(* IEC 61131-3 sources: 2026_Projet_YGO_ExcavatriceDragage/CODE/CODEURS, 10 files *)

(* ---- ST_Encoder_Calib.st ---- *)
(* ═══════════════════════════════════════════════════════════════
   🧲 ST_Encoder_Calib — Calibration & référence codeur (1 par treuil, RETAIN)
   ───────────────────────────────────────────────────────────────
   📄 Doc métier : DOC/AF/AF_Partie-09_Fonction_Encoder_v2.1.md
                   DOC/AF/AF_Partie-03_Contrats_Composants_v2.1.md
   🎛️ Une instance RETAIN par treuil (M1_EncoderCalib / M2_EncoderCalib).
   ═══════════════════════════════════════════════════════════════ *)

TYPE ST_Encoder_Calib :
STRUCT
    HomingRefRaw                  : UDINT;   // Valeur brute figée au dernier homing réussi
    LastKnownRawPos                : UDINT;   // Dernier point brut valide connu (§3.7, continu)
    RestartCoherenceTolerancePts    : UDINT := 1000;  // Tolérance redémarrage (~12% PointsPerRev 8192)
    Homed                          : BOOL;    // TRUE dès qu'un référencement a réussi
    HomingSuspect                  : BOOL;    // TRUE si incohérence détectée au redémarrage (§3.7)
END_STRUCT
END_TYPE

(* ---- ST_EncoderCalib.st ---- *)
(* ═══════════════════════════════════════════════════════════════
   🧲 ST_EncoderCalib — Calibration/référence codeur (1 par treuil, RETAIN)
   ───────────────────────────────────────────────────────────────
   📄 Doc métier : DOC/AF_Partie-09_Fonction_Encoder_Homing_v2.0.md §9
   🎛️ Une instance RETAIN par treuil (M1_EncoderCalib / M2_EncoderCalib).
   ⚠️ Ce lot (acquisition + mise à l'échelle) : `HomingRefRaw` reste
      modifiable MANUELLEMENT (RETAIN, valeur de test) tant que
      `FB_Encoder_Homing` (qui l'écrit normalement, §5) n'est pas codé —
      même principe que le stub GVL du lot Winch.
   ═══════════════════════════════════════════════════════════════ *)

TYPE ST_EncoderCalib :
STRUCT
    HomingRefRaw                  : UDINT;   // Valeur brute figée au dernier homing réussi
    LastKnownRawPos                : UDINT;   // Dernier point brut valide connu (§3.7, continu)
    RestartCoherenceTolerancePts    : UDINT := 1000;  // Tolérance redémarrage (~12% PointsPerRev 8192)
    Homed                          : BOOL;    // TRUE dès qu'un référencement a réussi
    HomingSuspect                  : BOOL;    // TRUE si incohérence détectée au redémarrage (§3.7)
END_STRUCT
END_TYPE

(* ---- ST_EncoderMeasurement.st ---- *)
(* ═══════════════════════════════════════════════════════════════
   📏 ST_EncoderMeasurement — Mesures codeur qualifiées (1 sous-DUT par treuil)
   ───────────────────────────────────────────────────────────────
   📄 Lot M1 · Doc : DOC/AF_Partie-06_Acquisition_Qualification_IO_v2.0.md §2ter
   🎨 Facts de la chaîne de mesure pure : Abs → Scale → Safety → SpeedMeasure.
   🔗 Producteur : PRG_02_Acquisition_CFC (chaîne codeur du treuil concerné).
   ✅ Tout BOOL = TRUE état normalisé. Aucun brut EtherCAT (alarmes/warnings,
      DEVICE_STATE) : ils restent exposés via ST_EncoderHMI (Supervision).
   ═══════════════════════════════════════════════════════════════ *)
TYPE ST_EncoderMeasurement :
STRUCT
    RawPos           : UDINT; (* Position brute codeur — gelée si EncoderAvailable=FALSE *)
    EncoderAvailable : BOOL;  (* TRUE = bus/esclave opérationnel *)
    CablePosM        : REAL;  (* Position câble (m, signée, + enroulé) *)
    CablePosMSafe    : REAL;  (* Position câble bornée [-99;+99] m — gelée sur doute *)
    EncoderIncoherent: BOOL;  (* TRUE = incohérence redémarrage → refuse SEMI_AUTO *)
    Speed_Mps        : REAL;  (* Vitesse absolue (m/s) — 0.0 si SpeedValid=FALSE *)
    SignedSpeed_Mps  : REAL;  (* Vitesse signée (m/s, + montée) — 0.0 si SpeedValid=FALSE *)
    SpeedValid       : BOOL;  (* TRUE si ≥ 6 éch. couvrant 50 ms *)
END_STRUCT
END_TYPE

(* ---- ST_EncoderMeasurements.st ---- *)
(* ═══════════════════════════════════════════════════════════════
   📏 ST_EncoderMeasurements — Mesures codeurs M1/M2 (contrat frontière)
   ───────────────────────────────────────────────────────────────
   📄 Lot M1 · Doc : DOC/AF/AF_Partie-06_Acquisition_Qualification_IO_v2.1.md §2ter
   🎨 Un sous-DUT par treuil (M1, M2) de la chaîne de mesure pure.
   🔗 Producteur unique : PRG_02_Acquisition_CFC (rang 02, chaîne codeur M1/M2).
      Lecteurs : PRG_04_Treuils_Benne_CFC, PRG_03_Modes_Cycle_CFC, Supervision/IHM.
   🛡️ Sans simulation : M1 reflète COD1, M2 reflète COD2 — jamais croisés.
   ═══════════════════════════════════════════════════════════════ *)
TYPE ST_EncoderMeasurements :
STRUCT
    M1 : ST_EncoderMeasurement; (* Chaîne de mesure treuil M1 (COD1) *)
    M2 : ST_EncoderMeasurement; (* Chaîne de mesure treuil M2 (COD2) *)
END_STRUCT
END_TYPE

(* ---- FB_Encoder_Abs.st ---- *)
(* ═══════════════════════════════════════════════════════════════
   🧲 FB_Encoder_Abs — Acquisition codeur absolu (accès bus, 1 responsabilité)
   ───────────────────────────────────────────────────────────────
   📄 Doc métier : DOC/AF_Partie-09_Fonction_Encoder_Homing_v2.0.md §3/§6
   ⚠️ RÉÉCRITURE COMPLÈTE (remplace la version legacy du projet, dossier
      CODEUR) : l'ancienne version utilisait `HomingTrigger` (recalage
      instantané par simple offset) + un mode `Teach` auto-calibré —
      **incompatibles** avec le design Partie10 (preset SDO avec
      accusé, formule `CableM_PerRev` fixe). Retirés : `HomingTrigger`,
      `WaterLevelOffset`, `TeachActive/StartRaw/EndRaw/RealDistance`.
   🧩 1 FB = 1 responsabilité : accès bus EtherCAT + séquence d'écriture
      preset. N'orchestre PAS le homing lui-même (ça sera le rôle de
      `FB_Encoder_Homing`, pas codé ce lot) — `PresetRequest`/`PresetValue`
      sont pilotés en dur (`FALSE`/`0`) dans `PRG_MAIN` pour l'instant.
   🧊 Principe « geler sur doute » (§6) : `RawPos`/`AngleRaw`/`TurnCount`
      ne sont PAS mis à jour si `EncoderAvailable = FALSE` — ils
      conservent leur dernière valeur plausible.
   ✅ SÉQUENCE PRESET (§5) — CONFIRMÉ TERRAIN 2026-07-02 : `PresetTriggerCmd := 2`
      (valeur de commande, pas un masque de bits) déclenche le
      référencement du codeur à `PresetValueOut`. `CodeSeqTriggerCmd`
      (canal réel `COD1_CodeSeqTrigCmd`) reste `0`, rôle **non identifié**
      (même par l'utilisateur/terrain) — ne jamais lui donner une valeur
      arbitraire tant que sa fonction n'est pas confirmée.
   🔴 PERTE DE FONCTION SIGNALÉE : l'ancienne version composait
      `FB_Encoder_Safety` en interne (survitesse via `In_SpdValue`).
      Ce n'est PAS repris ici (Partie10 ne le demande pas, hors
      périmètre du document) — `FB_Encoder_Safety` (overspeed) devient
      orphelin tant qu'un lot dédié ne décide pas de son sort (fusion
      avec le "saut incohérent" Partie10 §3.5, ou reprise telle quelle).
   🔧 CORRECTIF (2026-07-03, retour terrain) : `InvertDirection` **retiré**.
      Confirmé terrain : l'objet CoE `6000h` (bit0 : 4→5) inverse le sens
      de comptage **côté codeur** (F58x8 Kübler), configuré en **Startup
      Parameter** CODESYS (init automate) — pas un paramètre PLC. L'ancien
      calcul logiciel (`16#FFFFFFFF - RawPosIn`) était de toute façon
      **buggé** : il inversait sur toute la plage `UDINT` (32 bits) au
      lieu de la plage réelle du codeur (25 bits, `PointsPerRev ×
      MultiTurnRevsMax`), produisant des positions incohérentes après
      homing. Voir Partie10 §3bis.
   ═══════════════════════════════════════════════════════════════ *)

// === DECLARATION (à coller dans la partie déclaration du POU FB_Encoder_Abs) ===

FUNCTION_BLOCK PUBLIC FB_Encoder_Abs
VAR_INPUT
    Enable              : BOOL;        // Standard
    Reset               : BOOL;        // Acquittement défaut (front)
    PowerContactorEngaged     : BOOL;        // Standard
    Mode                : E_Mode;      // Standard (contexte, pas encore exploité ce lot)
    RawPosIn            : UDINT;       // Brut EtherCAT (ex. COD1_PosValue, %ID)
    AlarmsIn            : UINT;        // Brut EtherCAT (ex. COD1_Alarms)
    WarningsIn          : UINT;        // Brut EtherCAT (ex. COD1_Warnings) — informatif seulement
    SlaveOperational    : BOOL;        // FB_DiagEthercat — esclave EtherCAT opérationnel
    PointsPerRev        : UDINT := 8192;  // Résolution codeur confirmée (Partie10 §3.3)
    PresetRequest       : BOOL;        // Front — piloté par FB_Encoder_Homing via PRG_02_Encoders
    PresetValue         : UDINT;       // Cible brute — piloté par FB_Encoder_Homing (stub 0 ce lot)
    PresetTimeout       : TIME := T#2s;
    PresetTolerancePts  : UDINT := 10; // Tolérance relecture post-preset
END_VAR
VAR_OUTPUT
    Ready               : BOOL;
    Busy                : BOOL;
    Done                : BOOL;
    Error               : BOOL;
    ErrorId             : WORD;        // bit0: "Défaut communication codeur" - alarme/bus codeur ; bit1: "Erreur référencement (timeout)" - preset refusé/timeout
    State               : E_State;
    StateAtError        : E_State;
    RawPos              : UDINT;       // Position brute — GELÉE si EncoderAvailable=FALSE
    EncoderAvailable    : BOOL;
    AngleRaw            : UINT;        // Informatif maintenance : RawPos MOD PointsPerRev
    TurnCount           : UDINT;       // Informatif maintenance : RawPos / PointsPerRev
    PresetAck           : BOOL;        // Pulse 1 cycle — écriture confirmée
    PresetNak           : BOOL;        // Pulse 1 cycle — écriture refusée/timeout
    PresetTriggerCmd    : WORD;        // → à câbler sur COD_PresettTrigCmd (RxPDO)
    CodeSeqTriggerCmd   : WORD;        // → à câbler sur COD_CodeSeqTrigCmd (RxPDO)
    PresetValueOut      : UDINT;       // → à câbler sur COD_PresetValue (RxPDO)
END_VAR
VAR
    ResetEdge           : R_TRIG;
    ErrorEdge           : R_TRIG;
    PresetReqEdge       : R_TRIG;
    PresetTimer         : TON;
    PresetSeqStep       : INT;         // 0=IDLE, 1=pulse CodeSeq, 2=pulse Trig, 3=attente confirmation
    RawDiff             : DINT;
    PresetTimerVisual   : TON;         // Timer pour laisser le temps de voir l'impulsion (1.5s)
END_VAR

// === IMPLEMENTATION (à coller dans le corps ST du POU FB_Encoder_Abs) ===

// 🛑 1. GATE
IF NOT Enable THEN
    EncoderAvailable := FALSE;
    State := E_State.DISABLED;
    Ready := FALSE; Busy := FALSE; Done := FALSE;
    PresetTriggerCmd := 16#0000; CodeSeqTriggerCmd := 16#0000; PresetValueOut := 0;
    PresetSeqStep := 0;
    PresetTimer(IN := FALSE, PT := PresetTimeout);
    PresetTimerVisual(IN := FALSE, PT := T#500MS);
    RETURN;
END_IF;

Ready := TRUE;
State := E_State.READY;

// 🔑 2. RESET FRONT
ResetEdge(CLK := Reset);

// 🔍 3. DIAGNOSTIC BUS / ALARME
IF (AlarmsIn <> 0) OR NOT SlaveOperational THEN
    ErrorId := ErrorId OR 16#0001;
ELSE
    ErrorId := ErrorId AND 16#FFFE; (* Auto-clearing dès que le bus et l'esclave sont OK *)
END_IF;
EncoderAvailable := (ErrorId AND 16#0001) = 0;

// 📥 4. LECTURE POSITION — GELER SUR DOUTE (Partie10 §6)
// Si EncoderAvailable=FALSE : RawPos/AngleRaw/TurnCount conservent leur dernière valeur (pas de RETURN
// global ici pour ne pas geler aussi la séquence preset/l'état — seule la lecture est gelée).
IF EncoderAvailable THEN
    RawPos := RawPosIn;   // 🔧 2026-07-03 : sens de comptage géré côté codeur (CoE 6000h bit0,
                          // startup parameter CODESYS) — voir Partie10 §3bis. Plus de calcul ici.
    AngleRaw := UDINT_TO_UINT(RawPos MOD PointsPerRev);
    TurnCount := RawPos / PointsPerRev;
END_IF;

// 🔧 5. SÉQUENCE PRESET (écriture bus)
// ✅ Confirmé terrain (2026-07-02) : PresettTrigCmd := 2 déclenche le référencement à
//    PresetValue (valeur de commande, pas un masque de bits — corrige l'hypothèse initiale).
// 🔴 CodeSeqTrigCmd : rôle NON identifié (même par l'utilisateur/terrain) — laissé à 0,
//    PAS piloté tant que sa fonction n'est pas confirmée (fiche technique ou essai dédié).
//    Ne jamais lui donner une valeur arbitraire "au cas où".
PresetReqEdge(CLK := PresetRequest);
PresetAck := FALSE; PresetNak := FALSE; // pulses 1 cycle uniquement
CodeSeqTriggerCmd := 16#0000;           // 🔴 non piloté — rôle inconnu, voir note ci-dessus
CASE PresetSeqStep OF
    0: // IDLE
        PresetTriggerCmd := 0;
        IF PresetReqEdge.Q AND EncoderAvailable THEN
            PresetValueOut := PresetValue;
            PresetSeqStep := 1;
            PresetTimer(IN := TRUE, PT := PresetTimeout);
        END_IF;
    1: // Déclenchement preset (laissé actif pendant 0.5s pour confort visuel en simulation/bus)
        PresetTriggerCmd := 2;   // ✅ Valeur confirmée terrain — référence le codeur à PresetValueOut
        RawDiff := UDINT_TO_DINT(RawPos) - UDINT_TO_DINT(PresetValueOut);
        IF ABS(RawDiff) <= UDINT_TO_DINT(PresetTolerancePts) THEN
            PresetTimer(IN := FALSE, PT := PresetTimeout);
            PresetTimerVisual(IN := TRUE, PT := T#500MS);
            IF PresetTimerVisual.Q THEN
                PresetTriggerCmd := 0;
                PresetAck := TRUE;
                PresetSeqStep := 0;
                PresetTimerVisual(IN := FALSE, PT := T#500MS);
            END_IF;
        ELSIF PresetTimer.Q THEN
            PresetTriggerCmd := 0;
            PresetNak := TRUE;
            ErrorId := ErrorId OR 16#0002;
            PresetSeqStep := 0;
            PresetTimer(IN := FALSE, PT := PresetTimeout);
            PresetTimerVisual(IN := FALSE, PT := T#500MS);
        END_IF;
END_CASE;
IF ResetEdge.Q AND (PresetSeqStep = 0) THEN
    ErrorId := ErrorId AND 16#FFFD;
END_IF;

// 🧾 6. ERROR / STATEATERROR
Error := (ErrorId <> 16#0000);
ErrorEdge(CLK := Error);
IF ErrorEdge.Q THEN
    StateAtError := State;
END_IF;

Busy := (PresetSeqStep <> 0);
Done := PresetAck;

(* ---- FB_Encoder_Homing.st ---- *)
(* ═══════════════════════════════════════════════════════════════
   🎯 FB_Encoder_Homing — Référencement codeur nominal ou unitaire MAINT_N2
   ───────────────────────────────────────────────────────────────
   📄 Doc métier : DOC/AF_Partie-09_Fonction_Encoder_Homing_v2.0.md §1/§5/§7bis
   ⚠️ PÉRIMÈTRE : flux nominal (capteur haut + cible paramétrable) ou
      unitaire MAINT_N2 (treuil sélectionné + cible libre). Aucun mouvement
      moteur n'est piloté ici.
   🔌 PAS un FB de mouvement (Partie3 §1bis) : il n'écrit qu'une valeur
      de calibration, le treuil étant déjà à l'arrêt confirmé. Pas de
      `StartStop`/`SafeStop`.
   🧮 Calcul (généralise le cas historique cible=0.00, Partie10 §3.2/§3.3) :
      - `PresetValue` = `HomingRefTargetNominal` = (PointsPerRev × MultiTurnRevsMax) / 2
        (constante, TOUJOURS la même — centre exact de la plage, marge anti-débordement)
      - `HomingRefRaw` = `PresetValue` − round(`CfgTopSensorPosM` × PointsPerRev / CableM_PerRev)
        (ainsi `CablePosM` = `CfgTopSensorPosM` exactement au moment du homing)
      ⚠️ ÉVOLUTION vs interface §5 d'origine : `HomingRefRaw` est ajouté en sortie explicite
      (le document original supposait implicitement `HomingRefRaw := PresetValue`, valable
      uniquement pour une cible à 0.00 — ne fonctionne plus avec une cible non nulle ≈8.50 m).
   🧊 `ST_EncoderCalib` géré en interne (`VAR RETAIN`) — expose `Homed`/`HomingSuspect`/
      `HomingRefRaw` en sortie pour les consommateurs (`FB_Encoder_Scale`).
   🔴 SIMPLIFICATIONS assumées pour ce lot (à documenter/lever plus tard si besoin) :
      - Les 2 instances (M1/M2) sont autonomes : le même bouton IHM pilote les deux `Home`
        simultanément (câblage PRG_MAIN), mais chacune valide/rejette SES PROPRES conditions
        indépendamment (pas d'attente mutuelle ni de synchro de déclenchement).
      - `BtnConfirmCoherence`/§3.7 (incohérence redémarrage) : implémenté a minima (bit9), mais
        non testé en conditions réelles de coupure secteur — à revalider.
   ═══════════════════════════════════════════════════════════════ *)

// === DECLARATION (à coller dans la partie déclaration du POU FB_Encoder_Homing) ===

FUNCTION_BLOCK PUBLIC FB_Encoder_Homing
VAR_INPUT
    Enable               : BOOL;        // Standard
    Reset                : BOOL;        // Acquittement défaut (front) — bits 0/2/3/4/5 (voir §ErrorId)
    PowerContactorEngaged      : BOOL;        // Standard
    Mode                 : E_Mode;      // MAINT_N1 requis pour le flux nominal
    Home                 : BOOL;        // Demande de référencement (front, bouton IHM UNIQUE)
    UnitaryMode          : BOOL;        // TRUE = flux unitaire à cible libre (MAINT_N2 uniquement)
    WinchSelected        : BOOL;        // TRUE = cette instance est le treuil sélectionné
    CfgHomingTargetM        : REAL;        // Cible libre unitaire, limitée à [-99.0 ; +99.0] m
    BtnConfirmCoherence     : BOOL;        // Front — lève le doute §3.7 (bit9), sans réhoming complet
    TopPositionSensor    : BOOL;        // 🔧 2026-07-02 : capteur position haute UNIQUE, COMMUN aux 2 treuils
                                         // (les 2 câbles hissent ensemble le même ensemble mécanique) — câblé
                                         // IDENTIQUEMENT sur les instances M1 ET M2 (PAS un capteur par treuil),
                                         // voir PRG_MAIN.st
    CfgTopSensorPosM   : REAL := 8.5;   // Cible homing nominal (RETAIN site, voir Partie10 §7bis)
    FwdRevSpeedFeedbackOff : BOOL;      // 🔧 REX 2026-07-07 : retour unique "tous contacteurs sens+vitesse
                                         // retombés" CE TREUIL — arrêt confirmé (remplace ContactorFeedbackFwd/Rev)
    BrakeFeedback        : BOOL;        // Retour contacteur frein CE TREUIL (TRUE = relâché, FALSE = collé)
    RawPos               : UDINT;       // Sortie FB_Encoder_Abs (déjà gelée sur doute)
    EncoderAvailable     : BOOL;        // Sortie FB_Encoder_Abs
    PresetAck            : BOOL;        // Pulse — sortie FB_Encoder_Abs (écriture confirmée)
    PresetNak            : BOOL;        // Pulse — sortie FB_Encoder_Abs (écriture refusée/timeout)
    PointsPerRev         : UDINT := 8192;   // Confirmé fiche technique (Partie10 §3.3)
    MultiTurnRevsMax     : UDINT := 4096;   // Confirmé fiche technique (Partie10 §3.3)
    CableM_PerRev        : REAL := 2.0;     // Confirmé terrain 2026-07-02 (Partie10 §2)
    BypassGlobal         : BOOL := FALSE;   // 🌐 Ignore arrêt confirmé et capteur haut (mise en service)
END_VAR
VAR_OUTPUT
    Ready                : BOOL;
    Busy                 : BOOL;
    Done                 : BOOL;        // Pulse 1 cycle — référencement réussi (miroir PresetAck)
    Error                : BOOL;
    ErrorId              : WORD;        // Voir table de bits en en-tête de fichier / doc §5
    State                : E_State;
    StateAtError         : E_State;
    PresetRequest        : BOOL;        // Pulse → FB_Encoder_Abs.PresetRequest
    PresetValue          : UDINT;       // → FB_Encoder_Abs.PresetValue (= HomingRefTargetNominal)
    Homed                : BOOL;        // RETAIN interne, miroir Calib.Homed
    HomingSuspect        : BOOL;        // RETAIN interne, miroir Calib.HomingSuspect
    HomingRefRaw         : UDINT;       // RETAIN interne, miroir Calib.HomingRefRaw → FB_Encoder_Scale
END_VAR
VAR_IN_OUT
    Calib                : ST_EncoderCalib;   // Référence vers l'état persistant global (survit aux téléchargements)
END_VAR
VAR
    ResetEdge            : R_TRIG;
    ErrorEdge            : R_TRIG;
    HomeEdge             : R_TRIG;
    ConfirmCoherenceEdge : R_TRIG;
    InitDone             : BOOL;        // Contrôle cohérence §3.7 fait une fois par session Enable
    ArretConfirme        : BOOL;
    PresetValueCalc      : UDINT;       // = HomingRefTargetNominal (constant tant que PointsPerRev/MultiTurnRevsMax fixes)
    TargetPoints         : DINT;        // Écart signé CfgTopSensorPosM → points, figé pendant la séquence
    TargetPositionM      : REAL;        // Cible retenue : nominale ou unitaire
    RawDiffRestart       : DINT;        // Écart |RawPos - LastKnownRawPos| au redémarrage (§3.7)
END_VAR

// === IMPLEMENTATION (à coller dans le corps ST du POU FB_Encoder_Homing) ===

// 🛑 1. GATE — neutralisation ; on continue toutefois d'exposer le dernier état RETAIN connu
// (FB_Encoder_Scale a besoin de HomingRefRaw même si ce FB est désactivé)
IF NOT Enable OR NOT PowerContactorEngaged THEN
    PresetRequest := FALSE;
    PresetValue := 0;
    State := E_State.DISABLED;
    Ready := FALSE; Busy := FALSE; Done := FALSE;
    InitDone := FALSE;   // Force un nouveau contrôle §3.7 à la prochaine activation
    Homed := Calib.Homed;
    HomingSuspect := Calib.HomingSuspect;
    HomingRefRaw := Calib.HomingRefRaw;
    RETURN;
END_IF;

Ready := TRUE;

// 🔑 2. FRONTS
ResetEdge(CLK := Reset);
HomeEdge(CLK := Home);
ConfirmCoherenceEdge(CLK := BtnConfirmCoherence);

// 🔍 3. COHÉRENCE AU REDÉMARRAGE (§3.7) — une fois par session Enable, dès que le codeur répond
IF NOT InitDone THEN
    State := E_State.INIT;
    IF EncoderAvailable THEN
        RawDiffRestart := UDINT_TO_DINT(RawPos) - UDINT_TO_DINT(Calib.LastKnownRawPos);
        IF Calib.Homed AND (ABS(RawDiffRestart) > UDINT_TO_DINT(Calib.RestartCoherenceTolerancePts)) THEN
            Calib.HomingSuspect := TRUE;
            ErrorId := ErrorId OR 16#0200;   // bit9 : incohérence codeur au redémarrage
        END_IF;
        InitDone := TRUE;
    END_IF;
ELSE
    IF State = E_State.INIT THEN State := E_State.READY; END_IF;
END_IF;

// ✅ 4. LEVÉE DU DOUTE (BtnConfirmCoherence, §3.7) — indépendant du Reset générique
IF ConfirmCoherenceEdge.Q AND (Mode = E_Mode.MAINT_N1 OR Mode = E_Mode.MAINT_N2) THEN
    Calib.HomingSuspect := FALSE;
    ErrorId := ErrorId AND 16#FDFF;   // efface bit9
END_IF;

// 🎯 5. DEMANDE DE RÉFÉRENCEMENT (flux nominal)
// 🛡️ Les cibles nominale et unitaire sont rejetées hors du domaine codeur sûr [-99.00;+99.00] m.
// 🔧 REX 2026-07-07 : FwdRevSpeedFeedbackOff remplace (NOT ContactorFeedbackFwd) AND (NOT ContactorFeedbackRev)
// 🌐 BypassGlobal = TRUE → on saute la vérification d'arrêt (mise en service)
ArretConfirme := BypassGlobal OR (FwdRevSpeedFeedbackOff AND BrakeFeedback);

PresetRequest := FALSE;   // Défaut chaque cycle — repose uniquement sur le front HomeEdge ci-dessous
IF HomeEdge.Q AND (State <> E_State.BUSY) THEN
    IF UnitaryMode THEN
        TargetPositionM := CfgHomingTargetM;
    ELSE
        TargetPositionM := CfgTopSensorPosM;
    END_IF;

    // ✅ Homing autorisé en MAINT_N1 et MAINT_N2 — interdit en SEMI_AUTO et en cycle AUTO
    // 🌐 BypassGlobal = TRUE → saute TOUTES les vérifications, force le homing
    IF BypassGlobal THEN
        // Force homing sans condition
        PresetValueCalc := (PointsPerRev * MultiTurnRevsMax) / 2;
        TargetPoints := REAL_TO_DINT(TargetPositionM * UDINT_TO_REAL(PointsPerRev) / CableM_PerRev);
        PresetValue := PresetValueCalc;
        PresetRequest := TRUE;
        State := E_State.BUSY;
    ELSIF (Mode <> E_Mode.MAINT_N1) AND (Mode <> E_Mode.MAINT_N2) THEN
        ErrorId := ErrorId OR 16#0001;        // bit0 : mode non autorisé (seulement MAINT N1/N2)
    ELSIF UnitaryMode AND (Mode <> E_Mode.MAINT_N2) THEN
        ErrorId := ErrorId OR 16#0001;
    ELSIF UnitaryMode AND NOT WinchSelected THEN
        ErrorId := ErrorId OR 16#0002;        // bit1 : mauvais treuil sélectionné
    ELSIF NOT EncoderAvailable THEN
        ErrorId := ErrorId OR 16#0008;        // bit3 : codeur indisponible
    ELSIF NOT ArretConfirme THEN
        ErrorId := ErrorId OR 16#0004;        // bit2 : arrêt non confirmé (contacteurs/frein)
    ELSIF (TargetPositionM < -99.0) OR (TargetPositionM > 99.0) THEN
        ErrorId := ErrorId OR 16#0010;        // bit4 : cible nominale/unitaire hors limites
    ELSIF NOT BypassGlobal AND NOT UnitaryMode AND (TargetPositionM <> 0.0) AND TopPositionSensor THEN
        ErrorId := ErrorId OR 16#0010;        // bit4 : capteur position haute non confirmé
    ELSE
        // ✅ Toutes conditions réunies : calcul de la cible brute et déclenchement
        ErrorId := ErrorId AND 16#FFC0;       // Nettoie les erreurs de rejet 0..5
        PresetValueCalc := (PointsPerRev * MultiTurnRevsMax) / 2;               // Centre exact (§3.3)
        TargetPoints := REAL_TO_DINT(TargetPositionM * UDINT_TO_REAL(PointsPerRev) / CableM_PerRev);
        PresetValue := PresetValueCalc;
        PresetRequest := TRUE;                // Pulse 1 cycle — FB_Encoder_Abs détecte le front lui-même
        State := E_State.BUSY;
    END_IF;
END_IF;

// ⏳ 6. SUIVI DE LA SÉQUENCE (BUSY → confirmation)
Done := FALSE;
IF State = E_State.BUSY THEN
    IF PresetAck THEN
        Calib.HomingRefRaw := DINT_TO_UDINT(UDINT_TO_DINT(PresetValueCalc) - TargetPoints);
        Calib.Homed := TRUE;
        Calib.HomingSuspect := FALSE;
        Calib.LastKnownRawPos := PresetValueCalc;
        Done := TRUE;
        State := E_State.READY;
        // 🔧 REX 2026-07-24 : Un homing réussi efface l'intégralité de ErrorId (y compris les anciens rejets 0..5 et le bit9)
        ErrorId := 16#0000;
    ELSIF PresetNak THEN
        ErrorId := ErrorId OR 16#0020;        // bit5 : preset refusé/timeout (voir FB_Encoder_Abs)
        State := E_State.READY;
    END_IF;
END_IF;

// 🧾 7. RESET (front) — efface les bits « dernière tentative rejetée » (pas de cause persistante
// à revérifier ici : le prochain Home réévalue toutes les conditions de zéro, voir §5)
IF ResetEdge.Q THEN
    ErrorId := ErrorId AND 16#FFC0;   // efface bits 0..5 (garde bit9, levé seulement par BtnConfirmCoherence/Home)
END_IF;

// 📤 8. SORTIES ÉTAT
Error := (ErrorId <> 16#0000);
ErrorEdge(CLK := Error);
IF ErrorEdge.Q THEN
    StateAtError := State;
END_IF;

// Mise à jour continue du point brut valide connu (hors séquence de homing elle-même)
IF EncoderAvailable AND (State <> E_State.BUSY) THEN
    Calib.LastKnownRawPos := RawPos;
END_IF;

Busy := (State = E_State.BUSY);
Homed := Calib.Homed AND NOT Calib.HomingSuspect; // 🆕 REX 2026-07-08 : Perd l'état homed si suspect (démarrage ou fonctionnement), restauré après BtnConfirmCoherence
HomingSuspect := Calib.HomingSuspect;
HomingRefRaw := Calib.HomingRefRaw;

(* ---- FB_Encoder_Safety.st ---- *)
(* ═══════════════════════════════════════════════════════════════
   🛡️ FB_Encoder_Safety — Bornage physique + relais incohérence redémarrage (1 par treuil)
   ───────────────────────────────────────────────────────────────
   📄 Doc métier : DOC/AF_Partie-10_Fonction_Encoder_Homing_v1.10.md §3.6/§3.7
   🔌 FB STANDARD (Partie3 §1bis) : pas un FB de mouvement, pas de StartStop/SafeStop.
   🎯 PÉRIMÈTRE CE LOT (répond à l'incident CablePosM≈4096m après reset RETAIN) :
      - §3.6 Bornage absolu [-99.00 ; +99.00] m : `CablePosM` hors plage → valeur
        jugée IMPOSSIBLE, sortie `CablePosMSafe` GELÉE sur dernière valeur plausible
        (principe « geler sur doute », §6), ErrorId bit0.
      - §3.7 Relais de `HomingSuspect` (déjà détecté par `FB_Encoder_Homing`, jamais
        consommé nulle part avant ce lot) : ErrorId bit1.
      - `EncoderIncoherent` (= Error) → consommé par `FB_Modes` pour REFUSER
        `SEMI_AUTO` (reste possible de travailler en MAINT_N1/N2 pour re-référencer,
        voir échange utilisateur — PAS de SafeStop ici, ne bloque jamais le mouvement).
   🔴 HORS PÉRIMÈTRE CE LOT (Partie10 §3.5, reporté) : détection de saut EN COURS
      D'EXPLOITATION (plausibilité vitesse codeur, calcul sur cycles EtherCAT 4ms) —
      lot dédié à part entière, pas fait ici.
   ═══════════════════════════════════════════════════════════════ *)

// === DECLARATION (à coller dans la partie déclaration du POU FB_Encoder_Safety) ===

FUNCTION_BLOCK PUBLIC FB_Encoder_Safety
VAR_INPUT
    Enable           : BOOL;        // Standard
    Reset            : BOOL;        // Acquittement défaut (front) — bit0 uniquement (bit1 suit HomingSuspect, voir §7bis)
    EmergencyStopOk  : BOOL;        // Standard
    Mode             : E_Mode;      // Standard (contexte, pas encore exploité ce lot)
    CablePosM        : REAL;        // Sortie FB_Encoder_Scale DE CE TREUIL
    HomingSuspect    : BOOL;        // Sortie FB_Encoder_Homing DE CE TREUIL (§3.7, déjà calculé)
    PositionMinM     : REAL := -99.0;  // Bornage physique dur (Partie10 §3.6)
    PositionMaxM     : REAL := 99.0;
END_VAR
VAR_OUTPUT
    Ready            : BOOL;
    Busy             : BOOL;
    Done             : BOOL;
    Error            : BOOL;
    ErrorId          : WORD;        // bit0: "Position câble hors plage" - position hors plage physique ; bit1: "Incohérence position boot" - incohérence redémarrage (miroir HomingSuspect)
    State            : E_State;
    StateAtError     : E_State;
    CablePosMSafe    : REAL;        // CablePosM gelée sur dernière valeur plausible si hors plage
    EncoderIncoherent: BOOL;        // = Error — consommé par FB_Modes (refuse SEMI_AUTO)
END_VAR
VAR
    ResetEdge             : R_TRIG;
    ErrorEdge             : R_TRIG;
    LastPlausibleCablePosM: REAL;
END_VAR

// === IMPLEMENTATION (à coller dans le corps ST du POU FB_Encoder_Safety) ===

// 🛑 1. GATE — expose la dernière valeur plausible connue même désactivé
IF NOT Enable THEN
    Ready := FALSE; Busy := FALSE; Done := FALSE;
    State := E_State.DISABLED;
    CablePosMSafe := LastPlausibleCablePosM;
    EncoderIncoherent := FALSE;
    RETURN;
END_IF;

Ready := TRUE;
State := E_State.READY;

// 🔑 2. RESET FRONT
ResetEdge(CLK := Reset);

// 🔍 3. BORNAGE PHYSIQUE ABSOLU (§3.6) — bit0
IF (CablePosM < PositionMinM) OR (CablePosM > PositionMaxM) THEN
    ErrorId := ErrorId OR 16#0001;
ELSIF ResetEdge.Q THEN
    ErrorId := ErrorId AND 16#FFFE;
END_IF;

// 🔍 4. RELAIS INCOHÉRENCE REDÉMARRAGE (§3.7, calculée par FB_Encoder_Homing) — bit1
// Pas d'acquittement ici : la levée se fait via BtnConfirmCoherence/nouveau Home côté
// FB_Encoder_Homing (source), ce FB ne fait QUE relayer l'information pour FB_Modes.
IF HomingSuspect THEN
    ErrorId := ErrorId OR 16#0002;
ELSE
    ErrorId := ErrorId AND 16#FFFD;
END_IF;

// 🧊 5. GELER SUR DOUTE (§6) — CablePosMSafe ne suit PAS CablePosM si hors plage
IF (ErrorId AND 16#0001) = 16#0000 THEN
    LastPlausibleCablePosM := CablePosM;
END_IF;
CablePosMSafe := LastPlausibleCablePosM;

// 📤 6. SORTIES ÉTAT
Error := (ErrorId <> 16#0000);
ErrorEdge(CLK := Error);
IF ErrorEdge.Q THEN
    StateAtError := State;
END_IF;

EncoderIncoherent := Error;
Busy := FALSE;
Done := FALSE;

(* ---- FB_Encoder_Scale.st ---- *)
(* ═══════════════════════════════════════════════════════════════
   📏 FB_Encoder_Scale — Mise à l'échelle points → mètres (1 par treuil)
   ───────────────────────────────────────────────────────────────
   📄 Doc métier : DOC/AF_Partie-09_Fonction_Encoder_Homing_v2.0.md §2/§3.1
   ⚠️ RÉÉCRITURE (remplace la version legacy) : formule FIXE
      `CablePosM = (RawPos − HomingRefRaw) × (CableM_PerRev/PointsPerRev)`
      — retire le mode `Teach` auto-calibré (`EnableTeach`/`StartTeachPos`/
      `EndTeachPos`/`RealDistMeters`) : `CableM_PerRev` est un paramètre
      RETAIN fixe (site), pas recalculé dynamiquement (Partie10 §2).
   🧮 Arithmétique signée sûre (§3.1) : conversion en DINT AVANT la
      soustraction (jamais soustraire deux UDINT directement — un
      résultat négatif reboucle silencieusement vers ~2³²).
   🧩 Brique de calcul pure — pas de gel/bornage ici : `RawPos` en
      entrée est déjà gelé par `FB_Encoder_Abs` (§6) ; le bornage
      physique absolu [-99;+99] m est la responsabilité de
      `FB_Encoder_Safety` (§3.6, pas dans ce lot), pas de celle-ci.
   ═══════════════════════════════════════════════════════════════ *)

// === DECLARATION (à coller dans la partie déclaration du POU FB_Encoder_Scale) ===

FUNCTION_BLOCK PUBLIC FB_Encoder_Scale
VAR_INPUT
    RawPos          : UDINT;       // Position brute (sortie FB_Encoder_Abs, déjà gelée sur doute)
    HomingRefRaw    : UDINT;       // Référence brute figée au dernier homing (ST_EncoderCalib)
    CableM_PerRev   : REAL := 2.0; // Câble déroulé par tour (périmètre tambour confirmé 2026-07-02, réglable site)
    PointsPerRev    : UDINT := 8192; // Résolution codeur confirmée (Partie10 §3.3)
END_VAR
VAR_OUTPUT
    CablePosM       : REAL;        // Position câble en mètres, signée (+ enroulé, − sous l'eau)
END_VAR
VAR
    RawDiff         : DINT;        // Écart signé RawPos - HomingRefRaw (§3.1)
END_VAR

// === IMPLEMENTATION (à coller dans le corps ST du POU FB_Encoder_Scale) ===

// 🧮 Écart signé sûr : conversion DINT AVANT soustraction (§3.1) — jamais l'inverse
RawDiff := UDINT_TO_DINT(RawPos) - UDINT_TO_DINT(HomingRefRaw);

// 📏 Formule fixe points → mètres (Partie10 §2)
IF PointsPerRev > 0 THEN
    CablePosM := DINT_TO_REAL(RawDiff) * (CableM_PerRev / UDINT_TO_REAL(PointsPerRev));
ELSE
    CablePosM := 0.0;   // Garde division par zéro (PointsPerRev mal configuré)
END_IF;

(* ---- FB_Encoder_SpeedMeasure.st ---- *)
(* ═══════════════════════════════════════════════════════════════
   📐 FB_Encoder_SpeedMeasure — Mesure de vitesse câble horodatée
   ───────────────────────────────────────────────────────────────
   📄 Doc : DOC/AF_Partie-09_Fonction_Encoder_Homing_v2.0.md §3.8
   🛡️ Sécurité : mesure propriétaire de la chaîne codeur ; aucune réaction machine
   🧩 Dépendances : position sûre fournie par FB_Encoder_Safety
   ═══════════════════════════════════════════════════════════════ *)
FUNCTION_BLOCK PUBLIC FB_Encoder_SpeedMeasure
VAR_INPUT
    Enable        : BOOL; // Autorise l'acquisition
    Reset         : BOOL; // Purge immédiate de l'historique
    Position_M    : REAL; // Position câble sûre en mètres
    PositionValid : BOOL; // TRUE si la chaîne codeur garantit la position
END_VAR
VAR_OUTPUT
    Speed_Mps       : REAL; // Vitesse absolue sur la fenêtre horodatée
    SignedSpeed_Mps : REAL; // Vitesse signée : positive montée, négative descente
    Valid           : BOOL; // TRUE après 6 positions couvrant au moins 50 ms
END_VAR
VAR CONSTANT
    WindowTime   : TIME := T#50MS;
    SamplePeriod : TIME := T#10MS;
    SampleCount  : INT := 6;
END_VAR
VAR
    Positions_M : ARRAY[0..5] OF REAL;
    Timestamps  : ARRAY[0..5] OF TIME;
    CurrentTimestamp : TIME;
    LastTimestamp    : TIME;
    ElapsedSinceSample : TIME;
    WindowElapsed      : TIME;
    CollectedSamples   : INT;
    Index              : INT;
    TimestampInitialized : BOOL;
END_VAR

// ⏱️ Horodatage natif : le calcul utilise le temps réellement écoulé, jamais un cycle supposé.
CurrentTimestamp := TIME();

// 🧹 Toute rupture de confiance purge les six positions : aucune ancienne source ne peut contaminer la mesure.
IF NOT Enable OR Reset OR NOT PositionValid THEN
    Speed_Mps := 0.0;
    SignedSpeed_Mps := 0.0;
    Valid := FALSE;
    CollectedSamples := 0;
    TimestampInitialized := FALSE;
    RETURN;
END_IF;

// 🕒 Première position de la nouvelle fenêtre.
IF NOT TimestampInitialized THEN
    Positions_M[0] := Position_M;
    Timestamps[0] := CurrentTimestamp;
    LastTimestamp := CurrentTimestamp;
    CollectedSamples := 1;
    TimestampInitialized := TRUE;
    Speed_Mps := 0.0;
    SignedSpeed_Mps := 0.0;
    Valid := FALSE;
    RETURN;
END_IF;

// 🛡️ Rebouclage de TIME détecté localement : purge sans réutiliser le delta aberrant (indépendant de T88).
IF CurrentTimestamp < LastTimestamp THEN
    Positions_M[0] := Position_M;
    Timestamps[0] := CurrentTimestamp;
    LastTimestamp := CurrentTimestamp;
    CollectedSamples := 1;
    Speed_Mps := 0.0;
    SignedSpeed_Mps := 0.0;
    Valid := FALSE;
    RETURN;
END_IF;

ElapsedSinceSample := CurrentTimestamp - LastTimestamp;

// 🛡️ Delta nul : aucune division et aucun doublon d'échantillon.
IF ElapsedSinceSample <= T#0MS THEN
    RETURN;
END_IF;

// 📥 Six positions espacées d'au moins 10 ms donnent cinq intervalles sur la fenêtre interne de 50 ms.
IF ElapsedSinceSample >= SamplePeriod THEN
    LastTimestamp := CurrentTimestamp;

    IF CollectedSamples < SampleCount THEN
        Positions_M[CollectedSamples] := Position_M;
        Timestamps[CollectedSamples] := CurrentTimestamp;
        CollectedSamples := CollectedSamples + 1;
    ELSE
        FOR Index := 0 TO 4 DO
            Positions_M[Index] := Positions_M[Index + 1];
            Timestamps[Index] := Timestamps[Index + 1];
        END_FOR;
        Positions_M[5] := Position_M;
        Timestamps[5] := CurrentTimestamp;
    END_IF;

    IF CollectedSamples = SampleCount THEN
        // 🛡️ Ordre temporel et durée minimale contrôlés avant toute conversion/division.
        IF Timestamps[5] >= Timestamps[0] THEN
            WindowElapsed := Timestamps[5] - Timestamps[0];
            IF WindowElapsed >= WindowTime THEN
                SignedSpeed_Mps := (Positions_M[5] - Positions_M[0])
                                   / (UDINT_TO_REAL(TIME_TO_UDINT(WindowElapsed)) / 1000.0);
                Speed_Mps := ABS(SignedSpeed_Mps);
                Valid := TRUE;
            ELSE
                Speed_Mps := 0.0;
                SignedSpeed_Mps := 0.0;
                Valid := FALSE;
            END_IF;
        ELSE
            Speed_Mps := 0.0;
            SignedSpeed_Mps := 0.0;
            Valid := FALSE;
            CollectedSamples := 0;
            TimestampInitialized := FALSE;
        END_IF;
    END_IF;
END_IF;

(* ---- FB_Encoder_SpeedMonitor.st ---- *)
(* ═══════════════════════════════════════════════════════════════════════════════
   🔍 FB_Encoder_SpeedMonitor — Détection de variation brusque de vitesse câble
   ═══════════════════════════════════════════════════════════════════════════════
   📄 Brique standard de diagnostic — aucun pilotage moteur, aucun SafeStop.
   🎯 Compare deux mesures successives de vitesse linéaire câble en m/s.
   🧩 Le seuil et la durée de confirmation sont fournis par l'appelant :
      aucun réglage métier n'est figé dans cette brique.
   🛡️ Une variation confirmée pose ErrorId bit0. Le défaut reste mémorisé
      jusqu'à disparition de la cause et acquittement par front Reset.
   ═══════════════════════════════════════════════════════════════════════════════
   📄 Docs : DOC/AF_Partie-09_Fonction_Encoder_Homing_v2.0.md
*)

FUNCTION_BLOCK PUBLIC FB_Encoder_SpeedMonitor
VAR_INPUT
    Enable                     : BOOL;        // Autorise la surveillance
    Reset                      : BOOL;        // Acquittement par front
    PowerContactorEngaged            : BOOL;        // Contexte sécurité global valide
    Mode                       : E_Mode;      // Contexte de fonctionnement
    SpeedMps                   : REAL;        // Vitesse linéaire absolue mesurée (m/s)
    SpeedVariationThresholdMps : REAL;        // Variation minimale à surveiller (m/s)
    SpeedVariationTimeout      : TIME;        // Durée minimale de confirmation
    SpeedStabilityTimeout      : TIME;        // Durée sans variation avant vitesse stable
END_VAR
VAR_OUTPUT
    Ready                  : BOOL;
    Busy                   : BOOL;
    Done                   : BOOL;
    Error                  : BOOL;
    ErrorId                : WORD;        // bit0 : variation vitesse confirmée
    State                  : E_State;
    StateAtError           : E_State;
    SpeedDeltaMps          : REAL;        // Écart absolu entre deux mesures (m/s)
    SpeedVariationDetected : BOOL;        // Seuil dépassé sur le cycle courant
    SpeedVariationConfirmed: BOOL;        // Seuil dépassé pendant la durée requise
    SpeedStable            : BOOL;        // Vitesse stable pendant SpeedStabilityTimeout
END_VAR
VAR
    ResetEdge          : R_TRIG;
    ErrorEdge          : R_TRIG;
    VariationTimer     : TON;
    StabilityTimer     : TON;
    PreviousSpeedMps   : REAL;
    HasPreviousSpeed   : BOOL;
    VariationActive    : BOOL;
END_VAR

// 🛑 1. GATE — désactivation ou AU non réarmé : aucune alarme persistante.
IF NOT Enable OR NOT PowerContactorEngaged THEN
    Ready := FALSE;
    Busy := FALSE;
    Done := FALSE;
    Error := FALSE;
    ErrorId := 16#0000;
    State := E_State.DISABLED;
    SpeedDeltaMps := 0.0;
    SpeedVariationDetected := FALSE;
    SpeedVariationConfirmed := FALSE;
    SpeedStable := FALSE;
    VariationActive := FALSE;
    HasPreviousSpeed := FALSE;
    VariationTimer(IN := FALSE, PT := SpeedVariationTimeout);
    StabilityTimer(IN := FALSE, PT := SpeedStabilityTimeout);
    RETURN;
END_IF;

Ready := TRUE;
Busy := FALSE;
Done := FALSE;
State := E_State.READY;

// 🔑 2. RESET FRONT — l'acquittement n'efface le défaut que si la cause a disparu.
ResetEdge(CLK := Reset);

// 📏 3. CALCUL DE L'ÉCART DE VITESSE — première mesure utilisée comme référence.
IF NOT HasPreviousSpeed THEN
    PreviousSpeedMps := SpeedMps;
    HasPreviousSpeed := TRUE;
    SpeedDeltaMps := 0.0;
ELSE
    SpeedDeltaMps := ABS(SpeedMps - PreviousSpeedMps);
    PreviousSpeedMps := SpeedMps;
END_IF;

// 🔍 4. DÉTECTION BRUTE + FILTRE TEMPOREL — pas de déclenchement si la durée vaut zéro.
VariationActive := HasPreviousSpeed
                   AND (SpeedVariationThresholdMps >= 0.0)
                   AND (SpeedVariationTimeout > T#0ms)
                   AND (SpeedDeltaMps > SpeedVariationThresholdMps);
SpeedVariationDetected := VariationActive;

VariationTimer(IN := VariationActive, PT := SpeedVariationTimeout);
SpeedVariationConfirmed := VariationTimer.Q;
StabilityTimer(IN := HasPreviousSpeed AND NOT VariationActive AND (SpeedStabilityTimeout > T#0ms), PT := SpeedStabilityTimeout);
SpeedStable := StabilityTimer.Q;

IF SpeedVariationConfirmed THEN
    ErrorId := ErrorId OR 16#0001;
ELSIF ResetEdge.Q AND NOT VariationActive THEN
    ErrorId := ErrorId AND 16#FFFE;
END_IF;

// 📤 5. SORTIES D'ÉTAT — diagnostic standard, aucune commande mouvement.
Error := (ErrorId <> 16#0000);
ErrorEdge(CLK := Error);
IF ErrorEdge.Q THEN
    StateAtError := State;
END_IF;
